ABB RAPID module: Wobj_wobj_B.mod

MODULE Wobj_wobj_B
	! Points are read in order of declaration.
  ! Please do not change the order of points!

  LOCAL PERS robtarget pWobj_U_PointX1:=[[135.9564,-2147.717,-722.265],[0.000253810634603724,-0.727542340755463,0.686062157154083,0.000872761942446232],[-1,-1,2,0],[0,9E+09,9E+09,9E+09,9E+09,9E+09]];
	LOCAL PERS robtarget pWobj_U_PointX2:=[[430.8253,-2147.698,-722.2685],[0.000256351922871545,-0.727545082569122,0.686059236526489,0.000873812066856772],[-1,-1,2,0],[0,9E+09,9E+09,9E+09,9E+09,9E+09]];
	LOCAL PERS robtarget pWobj_U_PointY1:=[[461.318,-2036.453,-722.2611],[0.0002580912259873,-0.727556765079498,0.686046898365021,0.000879587489180267],[-1,-1,2,0],[0,9E+09,9E+09,9E+09,9E+09,9E+09]];

ENDMODULE
